{attribute 'qualified_only'}
//{attribute 'strict'}
TYPE E_MergeState :
(
	stStopped := 0,
	stClearTakeAway := 1,
	stMergeOperational := 2,
	stMergeManual := 3
)INT;
END_TYPE

(* stored: Version 1.1.0.1, ProductVersion 3.1.4024.4
   DUT E_MergeState: Id {5ab25a4f-a1e7-4478-82a6-f5ef67d6db7b} *)
